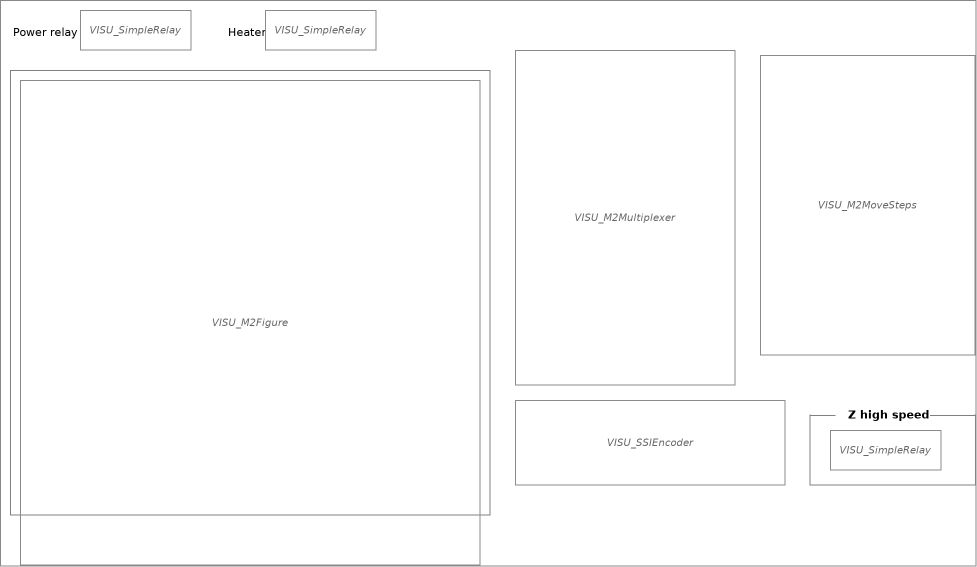
VISUALIZATION VISU_M2Technical  // 977x567
VAR_IN_OUT
	ref : M2;
    widget : M2Widget;
END_VAR
    Polyline (930,415) (975,415) (975,485) (810,485) (810,415) (835,415)
    Rectangle (10,70 480x445)
    Frame (20,80 460x485)
        shows VISU_M2Figure(ref := ref, widget := widget.figure)
    Frame (80,10 111x40)
        shows VISU_SimpleRelay(ref := ref.parts.powerRelay, widget := widget.powerRelay)
    Label (10,20 85x25), "Power relay"
    Frame (515,50 220x335)
        shows VISU_M2Multiplexer(ref := ref.parts.multiplexer, widget := widget.multiplexer)
    Frame (760,55 215x300)
        shows VISU_M2MoveSteps(ref_process := ref.processes.moveSteps, ref_procedure := ref.parts.moveStepsProcedure, widget := widget.moveSteps)
    Frame (515,400 270x85)
        shows VISU_SSIEncoder(ref := ref.parts.z.parts.encoder)
    Label (225,20 55x25), "Heater"
    Frame (265,10 111x40)
        shows VISU_SimpleRelay(ref := ref.parts.heater, widget := widget.heater)
    Frame (830,430 111x40)
        shows VISU_SimpleRelay(ref := ref.parts.z.parts.highSpeed, widget := widget.zHighSpeed)
    Label (845,405 90x20), "Z high speed"
END_VISUALIZATION

(* stored: Version 1.1.0.1, ProductVersion 3.1.4019.2
   Visu VISU_M2Technical: Id {0028ad04-11cf-4553-a2d0-16fd3100ecae} *)
